(* IEC 61131-3 sources: CodesysTest/export/UN00 - Sharp Bagger/EM01 - Bagger Head/CM05 - Printer/FB_BasicPrinter.pou/HasLabel.prop, 1 file *)

(* ---- Get.pm.st ---- *)
(*#-#-#-#-#-#-#-#-#-#---Declaration---#-#-#-#-#-#-#-#-#-#-#-#-#*)

VAR
END_VAR
(*#-#-#-#-#-#-#-#-#-#---Implementation---#-#-#-#-#-#-#-#-#-#-#-#-#*)

HasLabel := _hasLabel;
